FUNCTION_BLOCK IO_DO (* Digital output primitive; Backend 0 simulated, 1 GPIO (QX + GPIOChip handle), 2 Modbus CLIENT *)
  (* Standard: 61499-2 *)
  (* Version 2.0, 2026-09-27, Project contributors, Filling cell reference model *)
  PACKAGE fillingcell;
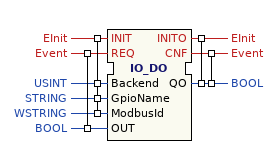
  EVENT_INPUT
    INIT : EInit WITH Backend, GpioName, ModbusId;
    REQ WITH OUT;
  END_EVENT
  EVENT_OUTPUT
    INITO : EInit WITH QO;
    CNF WITH QO;
  END_EVENT
  VAR_INPUT
    Backend : USINT;
    GpioName : STRING;
    ModbusId : WSTRING;
    OUT : BOOL;
  END_VAR
  VAR_OUTPUT
    QO : BOOL;
  END_VAR
  FBS
    Route : fillingcell::IO_RouteDO;
    Gpio : eclipse4diac::io::QX;
    Bus : iec61499::net::CLIENT_1_0;
  END_FBS
  EVENT_CONNECTIONS
    INIT TO Route.INIT;
    Route.INIT_IO TO Gpio.INIT;
    Gpio.INITO TO Bus.INIT;
    Bus.INITO TO Route.IO_READY;
    Route.INITO TO INITO;
    REQ TO Route.REQ;
    Route.REQ_G TO Gpio.REQ;
    Route.REQ_M TO Bus.REQ;
    Gpio.CNF TO Route.CNF_G;
    Bus.CNF TO Route.CNF_M;
    Route.CNF TO CNF;
  END_CONNECTIONS
  DATA_CONNECTIONS
    Backend TO Route.Backend;
    GpioName TO Gpio.PARAMS;
    ModbusId TO Bus.ID;
    Route.GQI TO Gpio.QI;
    Route.MQI TO Bus.QI;
    Gpio.QO TO Route.QO_G;
    Bus.QO TO Route.QO_M;
    Route.QO TO QO;
    OUT TO Route.OUT;
    Route.Value TO Gpio.OUT;
    Route.Value TO Bus.SD_1;
  END_CONNECTIONS
END_FUNCTION_BLOCK
